TYPE S_Hmi_Button :
STRUCT
	Click: BOOL;
	Enabled: BOOL;
	Led: BOOL;
END_STRUCT
END_TYPE

(* stored: Version 1.1.0.1, ProductVersion 3.1.4024.10
   DUT S_Hmi_Button: Id {bd5b506a-9540-4a0b-a5af-9f1eb2e250f3} *)
